TYPE ST_Genset_Get :
STRUCT
	CommunicationOK		: 	BOOL;
	FuelLow				: 	BOOL;
	FuelCritical		: 	BOOL;
		
	bGenBreakerClosed	:	BOOL;
	bMainBreakerClosed	:	BOOL;
	bGenRunning			:	BOOL;
	bGenVoltFreqOK		:	BOOL;
	bMainsFailure		:	BOOL;
	
	eActiveGenMode		:	eGenOperationMode;
	bIslandModeActive	:	BOOL;
	bAMFActive			:	BOOL;
	bPeakshaveActive	:	BOOL;
	bFixedPowerActive	:	BOOL;

	ar_LineVoltage	:	ARRAY[0..3] OF REAL;
	ar_PhaseVoltage	:	ARRAY[0..3] OF REAL;
	ar_Frequency	:	ARRAY[0..3] OF REAL;
	ar_Current		:	ARRAY[0..3] OF REAL;
	ar_PowerFactor	: 	ARRAY[0..0] OF REAL;
	ar_ActivePower 	:   ARRAY[0..3] OF REAL;
	ar_ReactivePower: 	ARRAY[0..0] OF REAL;
	ar_ApparentPower:	ARRAY[0..0] OF REAL;
	
	
END_STRUCT
END_TYPE

(* stored: Version 1.1.0.1, ProductVersion 3.1.4026.18
   DUT ST_Genset_Get: Id {bf3be5cf-87c4-4ac1-86be-7a59f6533efe} *)
